(*
version 1.1	2 okt 2006
programmer 	hugo
tested by	tobias

extracts the hour of a Time_of_day
*)
FUNCTION HOUR : INT
VAR_INPUT
	itod : TOD;
END_VAR

HOUR := DWORD_TO_INT(TOD_TO_DWORD(itod) / 3600000);


(* change history
hm 4. aug 2006	rev 1.0
	original version

hm 2.10.2006 	rev 1.1
	changed name of input to itod

*)

END_FUNCTION

(* stored: Version 1.1.0.1
   POU HOUR: Id {d65a0da1-ee08-47d2-bd66-1af974b46a10}, SpecialFunc None *)
